// TIA Portal V19 export
TYPE "DecoilersHRot_Status"
   STRUCT
      Rotation : "ValveMachine_COut";
      Pivot : "ValveMachine_COut";
      Traslation : "Positioning_DOL_Machine_COut";
      DecoilerX_InLine_CheckNext { S7_SetPoint := 'True'} : Bool;
      Decoiler1_InLine : Bool;
      Decoiler2_InLine : Bool;
      Translation_InPosition : Bool;
   END_STRUCT;
END_TYPE
